TYPE EKF_Data :
STRUCT
	State : state;
	wheelSpeed : ARRAY[1..3] OF LREAL;   (* w1,w2,w3 *)
	P_Start : ARRAY[1..9] OF LREAL;
	timestamp : LREAL;
END_STRUCT
END_TYPE

(* stored: Version 1.1.0.1, ProductVersion 3.1.4026.13
   DUT EKF_Data: Id {2b88a999-2f3a-4d36-b52e-5f3113db0285} *)
